FUNCTION_BLOCK SS5a_ps_Camera (* Composite FB wrapping other FBs *)
  (* Standard: 61499-2 *)
  (* Version 1.0, 2025-08-26, PS_Transformer_for_Unknown *)
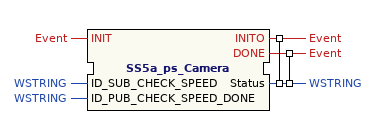
  EVENT_INPUT
    INIT; (* Initialization Request *)
  END_EVENT
  EVENT_OUTPUT
    INITO WITH Status; (* Initialization Confirm *)
    DONE WITH Status; (* Execution Confirmation *)
  END_EVENT
  VAR_INPUT
    ID_SUB_CHECK_SPEED : WSTRING;
    ID_PUB_CHECK_SPEED_DONE : WSTRING;
  END_VAR
  VAR_OUTPUT
    Status : WSTRING; (* Output event qualifier *)
  END_VAR
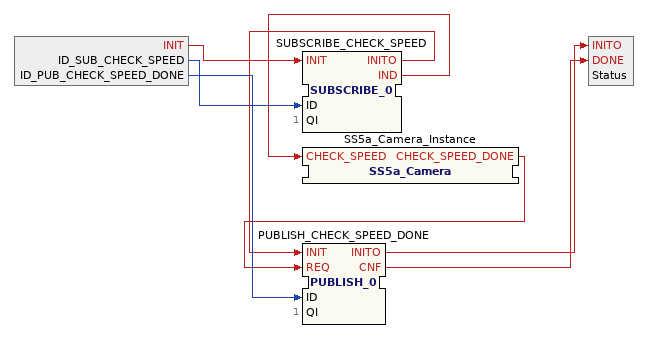
  FBS
    SS5a_Camera_Instance : SS5a_Camera;
    SUBSCRIBE_CHECK_SPEED : SUBSCRIBE_0(QI := 1);
    PUBLISH_CHECK_SPEED_DONE : PUBLISH_0(QI := 1);
  END_FBS
  EVENT_CONNECTIONS
    INIT TO SUBSCRIBE_CHECK_SPEED.INIT;
    SUBSCRIBE_CHECK_SPEED.INITO TO PUBLISH_CHECK_SPEED_DONE.INIT;
    PUBLISH_CHECK_SPEED_DONE.INITO TO INITO;
    SUBSCRIBE_CHECK_SPEED.IND TO SS5a_Camera_Instance.CHECK_SPEED;
    SS5a_Camera_Instance.CHECK_SPEED_DONE TO PUBLISH_CHECK_SPEED_DONE.REQ;
    PUBLISH_CHECK_SPEED_DONE.CNF TO DONE;
  END_CONNECTIONS
  DATA_CONNECTIONS
    ID_SUB_CHECK_SPEED TO SUBSCRIBE_CHECK_SPEED.ID;
    ID_PUB_CHECK_SPEED_DONE TO PUBLISH_CHECK_SPEED_DONE.ID;
  END_CONNECTIONS
END_FUNCTION_BLOCK
